Fanuc KAREL source: kt00475.KL

-- PROVISIONAL review KL for V1013-1; original PC SHA256 9c2e5306c295e74d43a96989c5423b5fca64aca1f0aef38046aa900a81088228
-- Incomplete behavior may be omitted. Consult companion uncertainty JSON. Do not deploy.
PROGRAM KT00475
%NOLOCKGROUP
-- UNRESOLVED_DECL P1 type=000101
-- UNRESOLVED_DECL P2 type=000101
-- UNRESOLVED_DECL OUT type=000102
BEGIN
  -- UNRESOLVED_PC offsets 5-34; opcodes 49,49,60,7E,4A
  -- UNRESOLVED_PC offsets 39-43; opcodes 7F
END KT00475
